{attribute 'GeneratedUsingTerminal: EL3311-0000-0018'}
{attribute addProperty BoxType "EL3311-0000-0018"}
{attribute addProperty Id "TC_InputsAT %I*TC_Inputs_4A3944819WcStateAT %I*WcState_9091E0EB2InfoDataAT %I*InfoData_32EB74EA10"}
{attribute addProperty CRC "713902466"}
{attribute addProperty Size "21"}
TYPE EL3311_2A8D4982 EXTENDS EtcSlaveTerminalBase_947E5A46 :
STRUCT
	{attribute addProperty Name "TC_Inputs"}
	TC_Inputs : TC_Inputs_4A394481;
	{attribute addProperty Name "WcState"}
	WcState : WcState_9091E0EB;
	{attribute addProperty Name "InfoData"}
	InfoData : InfoData_32EB74EA;
END_STRUCT
END_TYPE

(* stored: Version 1.2.0.0, ProductVersion 3.1.4024.9
   DUT EL3311_2A8D4982: Id {b2d71c62-76c9-41d0-af8c-669ca1011965} *)
